Staubli VAL3: clrscr.pgx

public program clrscr()
begin
  cls()
  title("")
end
